// Device/Application/visualization/baseModule/grd
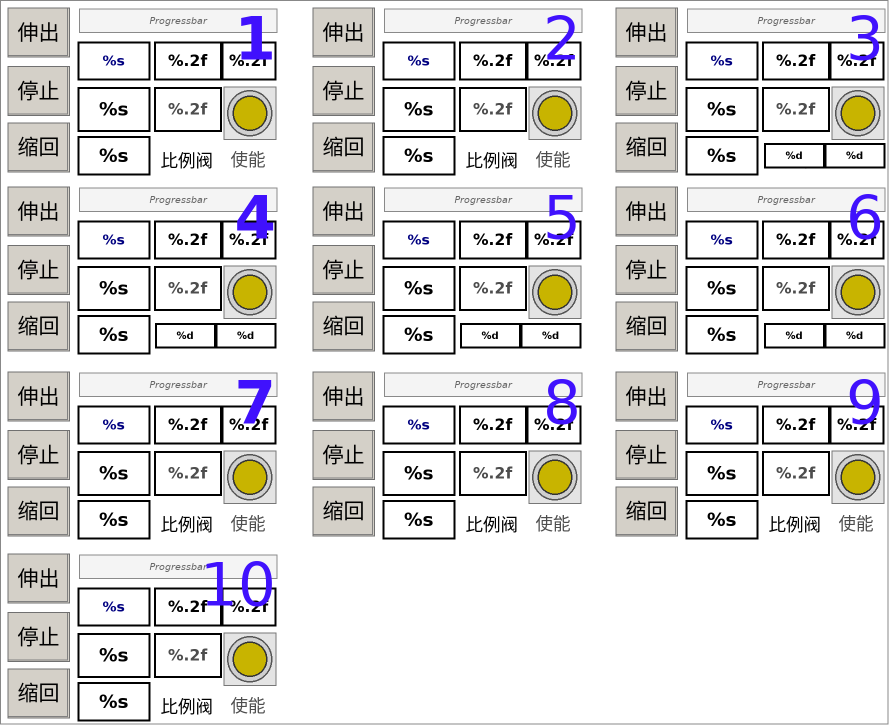
VISUALIZATION grd  // 889x725
    Frame (0,0 279x177), "1"
        shows DevUnit0(extendButton := gUI.grd[1].btnExtend, retractButton := gUI.grd[1].btnRetract, stopButton := gUI.grd[1].btnStop, percentShow := gUI.grd[1].extendPercent, nameShow := gUI.grd[1].name, wnameShow := gUI.grd[1].wname, hzname := gUI.grd[1].hzname, posShow := gUI.grd[1].postion, spdShow := gUI.grd[1].speed, pwrEnable := gUI.grd[1].pwrEnable, pwrPct := gUI.grd[1].pwrPercent)
    Frame (305,0 279x177), "2"
        shows DevUnit0(extendButton := gUI.grd[2].btnExtend, retractButton := gUI.grd[2].btnRetract, stopButton := gUI.grd[2].btnStop, percentShow := gUI.grd[2].extendPercent, nameShow := gUI.grd[2].name, wnameShow := gUI.grd[2].wname, hzname := gUI.grd[2].hzname, posShow := gUI.grd[2].postion, spdShow := gUI.grd[2].speed, pwrEnable := gUI.grd[2].pwrEnable, pwrPct := gUI.grd[2].pwrPercent)
    Frame (608,0 279x177), "3"
        shows DevUnit0(extendButton := gUI.grd[3].btnExtend, retractButton := gUI.grd[3].btnRetract, stopButton := gUI.grd[3].btnStop, percentShow := gUI.grd[3].extendPercent, nameShow := gUI.grd[3].name, wnameShow := gUI.grd[3].wname, hzname := gUI.grd[3].hzname, posShow := gUI.grd[3].postion, spdShow := gUI.grd[3].speed, pwrEnable := gUI.grd[3].pwrEnable, pwrPct := gUI.grd[3].pwrPercent)
    Frame (0,179 279x177), "4"
        shows DevUnit0(extendButton := gUI.grd[4].btnExtend, retractButton := gUI.grd[4].btnRetract, stopButton := gUI.grd[4].btnStop, percentShow := gUI.grd[4].extendPercent, nameShow := gUI.grd[4].name, wnameShow := gUI.grd[4].wname, hzname := gUI.grd[4].hzname, posShow := gUI.grd[4].postion, spdShow := gUI.grd[4].speed, pwrEnable := gUI.grd[4].pwrEnable, pwrPct := gUI.grd[4].pwrPercent)
    Frame (305,179 279x177), "5"
        shows DevUnit0(extendButton := gUI.grd[5].btnExtend, retractButton := gUI.grd[5].btnRetract, stopButton := gUI.grd[5].btnStop, percentShow := gUI.grd[5].extendPercent, nameShow := gUI.grd[5].name, wnameShow := gUI.grd[5].wname, hzname := gUI.grd[5].hzname, posShow := gUI.grd[5].postion, spdShow := gUI.grd[5].speed, pwrEnable := gUI.grd[5].pwrEnable, pwrPct := gUI.grd[5].pwrPercent)
    Frame (608,179 279x177), "6"
        shows DevUnit0(extendButton := gUI.grd[6].btnExtend, retractButton := gUI.grd[6].btnRetract, stopButton := gUI.grd[6].btnStop, percentShow := gUI.grd[6].extendPercent, nameShow := gUI.grd[6].name, wnameShow := gUI.grd[6].wname, hzname := gUI.grd[6].hzname, posShow := gUI.grd[6].postion, spdShow := gUI.grd[6].speed, pwrEnable := gUI.grd[6].pwrEnable, pwrPct := gUI.grd[6].pwrPercent)
    Frame (0,364 279x177), "7"
        shows DevUnit0(extendButton := gUI.grd[7].btnExtend, retractButton := gUI.grd[7].btnRetract, stopButton := gUI.grd[7].btnStop, percentShow := gUI.grd[7].extendPercent, nameShow := gUI.grd[7].name, wnameShow := gUI.grd[7].wname, hzname := gUI.grd[7].hzname, posShow := gUI.grd[7].postion, spdShow := gUI.grd[7].speed, pwrEnable := gUI.grd[7].pwrEnable, pwrPct := gUI.grd[7].pwrPercent)
    Frame (305,364 279x177), "8"
        shows DevUnit0(extendButton := gUI.grd[8].btnExtend, retractButton := gUI.grd[8].btnRetract, stopButton := gUI.grd[8].btnStop, percentShow := gUI.grd[8].extendPercent, nameShow := gUI.grd[8].name, wnameShow := gUI.grd[8].wname, hzname := gUI.grd[8].hzname, posShow := gUI.grd[8].postion, spdShow := gUI.grd[8].speed, pwrEnable := gUI.grd[8].pwrEnable, pwrPct := gUI.grd[8].pwrPercent)
    Frame (608,364 279x177), "9"
        shows DevUnit0(extendButton := gUI.grd[9].btnExtend, retractButton := gUI.grd[9].btnRetract, stopButton := gUI.grd[9].btnStop, percentShow := gUI.grd[9].extendPercent, nameShow := gUI.grd[9].name, wnameShow := gUI.grd[9].wname, hzname := gUI.grd[9].hzname, posShow := gUI.grd[9].postion, spdShow := gUI.grd[9].speed, pwrEnable := gUI.grd[9].pwrEnable, pwrPct := gUI.grd[9].pwrPercent)
    Frame (0,546 279x177), "10"
        shows DevUnit0(extendButton := gUI.grd[10].btnExtend, retractButton := gUI.grd[10].btnRetract, stopButton := gUI.grd[10].btnStop, percentShow := gUI.grd[10].extendPercent, nameShow := gUI.grd[10].name, wnameShow := gUI.grd[10].wname, hzname := gUI.grd[10].hzname, posShow := gUI.grd[10].postion, spdShow := gUI.grd[10].speed, pwrEnable := gUI.grd[10].pwrEnable, pwrPct := gUI.grd[10].pwrPercent)
    Frame (764,143 123x27)
        shows currentUnit(Ixt := gDev.grd[3].current[1], Irt := gDev.grd[3].current[2])
    Frame (155,323 123x27)
        shows currentUnit(Ixt := gDev.grd[4].current[1], Irt := gDev.grd[4].current[2])
    Frame (460,323 123x27)
        shows currentUnit(Ixt := gDev.grd[5].current[1], Irt := gDev.grd[5].current[2])
    Frame (764,323 123x27)
        shows currentUnit(Ixt := gDev.grd[6].current[1], Irt := gDev.grd[6].current[2])
END_VISUALIZATION

// Device/Application/visualization/baseModule/setting
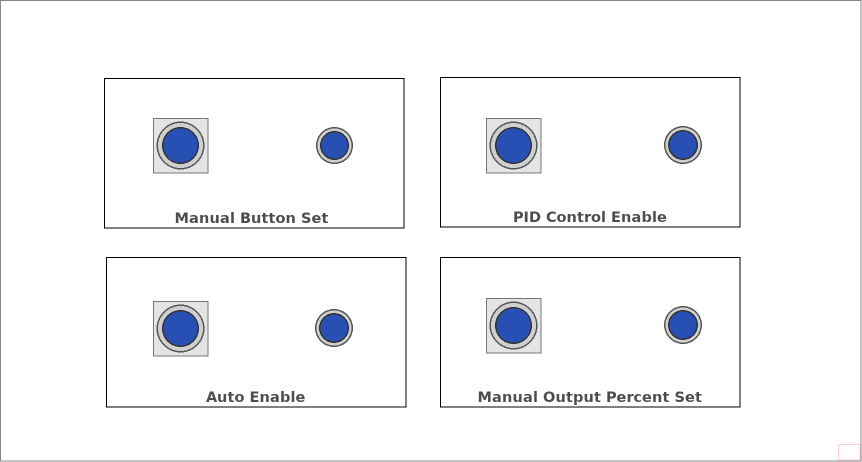
VISUALIZATION setting  // 862x462
    Rectangle (104,78 300x150), "Manual Button Set"
    Lamp1 (313,122 43x47), variable: gUI.mode.manualButtonSet, style: Lamp-Lamp1-Blue
    PushSwitchLed (153,113 55x65), variable: gUI.mode.manualButtonSet, behaviour: TOGGLE, style: Switch-PushSwitchLed-Blue
    Rectangle (440,77 300x150), "PID Control Enable"
    Lamp1 (661,122 44x46), variable: gUI.mode.usePID, style: Lamp-Lamp1-Blue
    PushSwitchLed (486,113 55x65), variable: gUI.mode.usePID, behaviour: TOGGLE, style: Switch-PushSwitchLed-Blue
    Rectangle (838,444 22x16)
    Group (106,257 300x150)
        Rectangle (0,0 300x150), "Auto Enable"
        Lamp1 (206,48 44x46), variable: gUI.mode.autoEnable, style: Lamp-Lamp1-Blue
        PushSwitchLed (47,39 55x65), variable: gUI.mode.autoEnable, behaviour: TOGGLE, style: Switch-PushSwitchLed-Blue
    Rectangle (440,257 300x150), "Manual Output Percent Set"
    Lamp1 (661,302 44x46), variable: gUI.mode.manualPercentSet, style: Lamp-Lamp1-Blue
    PushSwitchLed (486,293 55x65), variable: gUI.mode.manualPercentSet, behaviour: TOGGLE, style: Switch-PushSwitchLed-Blue
END_VISUALIZATION

// Device/Application/main
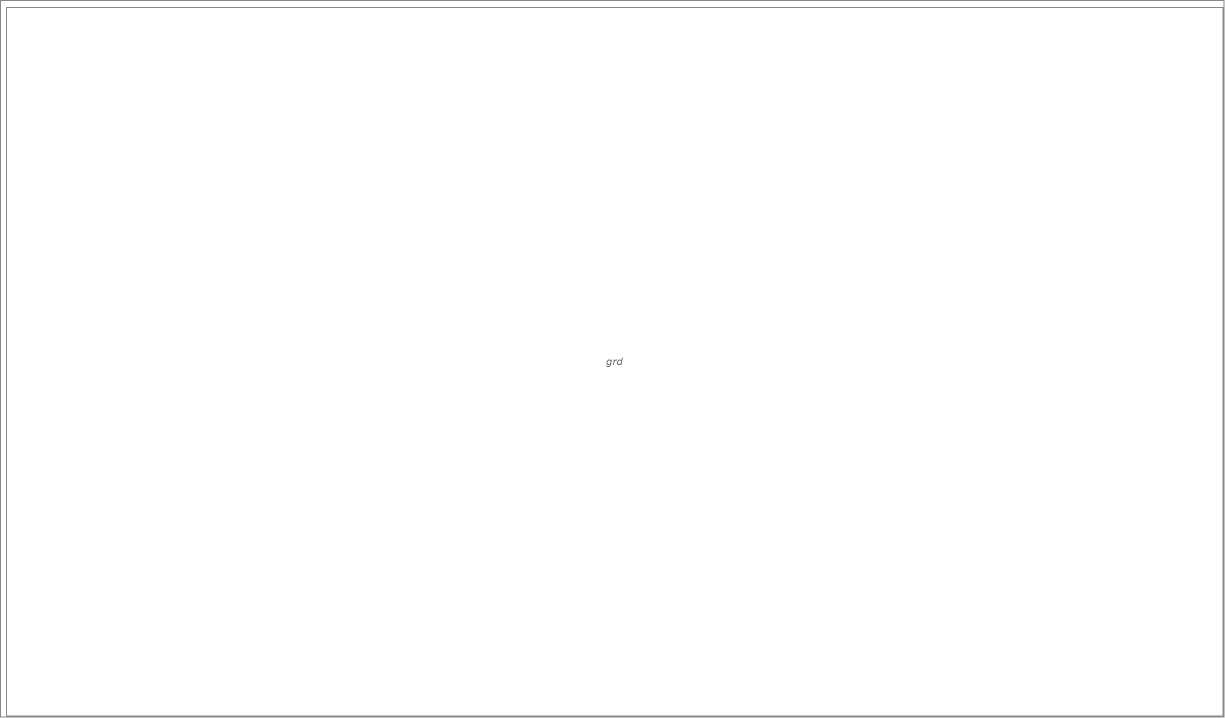
VISUALIZATION main  // 1225x718
    TabControl (6,7 1217x709)
        shows grd()
        shows sky()
        shows testPID()
        shows setting()
        [0]: ImageId=__VisualizationStyle.Element-Switch-PushSwitch-Green-On
        [1]: ImageId=__VisualizationStyle.Element-Switch-PushSwitch-Blue-On
        [2]: ImageId=__VisualizationStyle.Element-Switch-RotarySwitch-Blue-RightUp
        [3]: ImageId=__VisualizationStyle.Element-Switch-PushSwitch-Blue-On
END_VISUALIZATION

// Device/Application/visualization/baseModule/sky
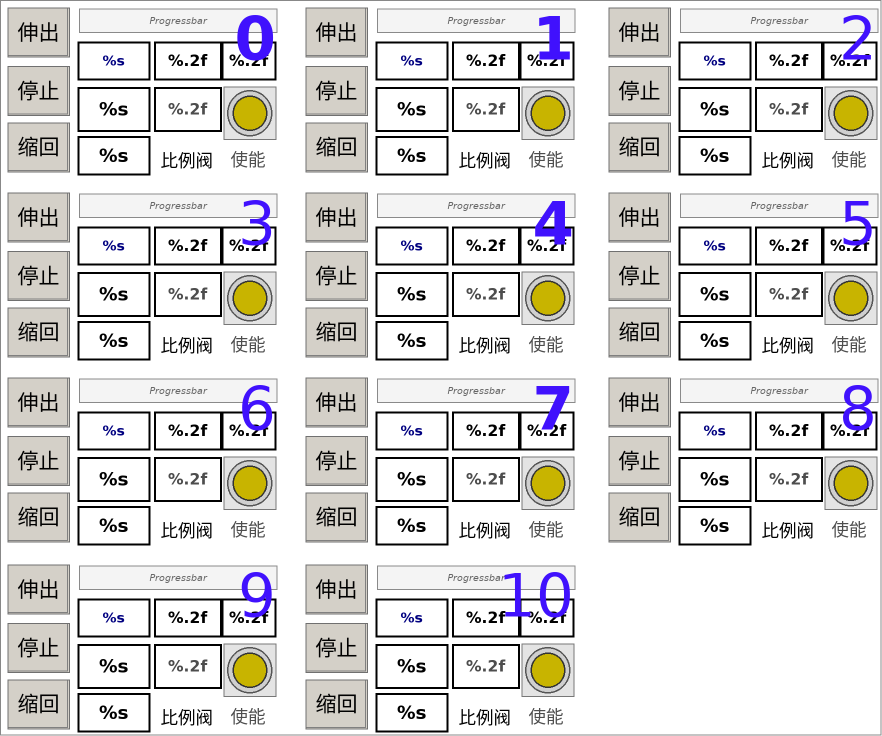
VISUALIZATION sky  // 882x736
    Frame (0,185 279x177), "3"
        shows DevUnit0(extendButton := gUI.sky[3].btnExtend, retractButton := gUI.sky[3].btnRetract, stopButton := gUI.sky[3].btnStop, percentShow := gUI.sky[3].extendPercent, nameShow := gUI.sky[3].name, wnameShow := gUI.sky[3].wname, hzname := gUI.sky[3].hzname, posShow := gUI.sky[3].postion, spdShow := gUI.sky[3].speed, pwrEnable := gUI.sky[3].pwrEnable, pwrPct := gUI.sky[3].pwrPercent)
    Frame (298,185 279x177), "4"
        shows DevUnit0(extendButton := gUI.sky[4].btnExtend, retractButton := gUI.sky[4].btnRetract, stopButton := gUI.sky[4].btnStop, percentShow := gUI.sky[4].extendPercent, nameShow := gUI.sky[4].name, wnameShow := gUI.sky[4].wname, hzname := gUI.sky[4].hzname, posShow := gUI.sky[4].postion, spdShow := gUI.sky[4].speed, pwrEnable := gUI.sky[4].pwrEnable, pwrPct := gUI.sky[4].pwrPercent)
    Frame (601,185 279x177), "5"
        shows DevUnit0(extendButton := gUI.sky[5].btnExtend, retractButton := gUI.sky[5].btnRetract, stopButton := gUI.sky[5].btnStop, percentShow := gUI.sky[5].extendPercent, nameShow := gUI.sky[5].name, wnameShow := gUI.sky[5].wname, hzname := gUI.sky[5].hzname, posShow := gUI.sky[5].postion, spdShow := gUI.sky[5].speed, pwrEnable := gUI.sky[5].pwrEnable, pwrPct := gUI.sky[5].pwrPercent)
    Frame (0,370 279x177), "6"
        shows DevUnit0(extendButton := gUI.sky[6].btnExtend, retractButton := gUI.sky[6].btnRetract, stopButton := gUI.sky[6].btnStop, percentShow := gUI.sky[6].extendPercent, nameShow := gUI.sky[6].name, wnameShow := gUI.sky[6].wname, hzname := gUI.sky[6].hzname, posShow := gUI.sky[6].postion, spdShow := gUI.sky[6].speed, pwrEnable := gUI.sky[6].pwrEnable, pwrPct := gUI.sky[6].pwrPercent)
    Frame (298,370 279x177), "7"
        shows DevUnit0(extendButton := gUI.sky[7].btnExtend, retractButton := gUI.sky[7].btnRetract, stopButton := gUI.sky[7].btnStop, percentShow := gUI.sky[7].extendPercent, nameShow := gUI.sky[7].name, wnameShow := gUI.sky[7].wname, hzname := gUI.sky[7].hzname, posShow := gUI.sky[7].postion, spdShow := gUI.sky[7].speed, pwrEnable := gUI.sky[7].pwrEnable, pwrPct := gUI.sky[7].pwrPercent)
    Frame (601,370 279x177), "8"
        shows DevUnit0(extendButton := gUI.sky[8].btnExtend, retractButton := gUI.sky[8].btnRetract, stopButton := gUI.sky[8].btnStop, percentShow := gUI.sky[8].extendPercent, nameShow := gUI.sky[8].name, wnameShow := gUI.sky[8].wname, hzname := gUI.sky[8].hzname, posShow := gUI.sky[8].postion, spdShow := gUI.sky[8].speed, pwrEnable := gUI.sky[8].pwrEnable, pwrPct := gUI.sky[8].pwrPercent)
    Frame (0,557 279x177), "9"
        shows DevUnit0(extendButton := gUI.sky[9].btnExtend, retractButton := gUI.sky[9].btnRetract, stopButton := gUI.sky[9].btnStop, percentShow := gUI.sky[9].extendPercent, nameShow := gUI.sky[9].name, wnameShow := gUI.sky[9].wname, hzname := gUI.sky[9].hzname, posShow := gUI.sky[9].postion, spdShow := gUI.sky[9].speed, pwrEnable := gUI.sky[9].pwrEnable, pwrPct := gUI.sky[9].pwrPercent)
    Frame (298,557 279x177), "10"
        shows DevUnit0(extendButton := gUI.sky[10].btnExtend, retractButton := gUI.sky[10].btnRetract, stopButton := gUI.sky[10].btnStop, percentShow := gUI.sky[10].extendPercent, nameShow := gUI.sky[10].name, wnameShow := gUI.sky[10].wname, hzname := gUI.sky[10].hzname, posShow := gUI.sky[10].postion, spdShow := gUI.sky[10].speed, pwrEnable := gUI.sky[10].pwrEnable, pwrPct := gUI.sky[10].pwrPercent)
    Frame (298,0 279x177), "1"
        shows DevUnit0(extendButton := gUI.sky[1].btnExtend, retractButton := gUI.sky[1].btnRetract, stopButton := gUI.sky[1].btnStop, percentShow := gUI.sky[1].extendPercent, nameShow := gUI.sky[1].name, wnameShow := gUI.sky[1].wname, hzname := gUI.sky[1].hzname, posShow := gUI.sky[1].postion, spdShow := gUI.sky[1].speed, pwrEnable := gUI.sky[1].pwrEnable, pwrPct := gUI.sky[1].pwrPercent)
    Frame (601,0 279x177), "2"
        shows DevUnit0(extendButton := gUI.sky[2].btnExtend, retractButton := gUI.sky[2].btnRetract, stopButton := gUI.sky[2].btnStop, percentShow := gUI.sky[2].extendPercent, nameShow := gUI.sky[2].name, wnameShow := gUI.sky[2].wname, hzname := gUI.sky[2].hzname, posShow := gUI.sky[2].postion, spdShow := gUI.sky[2].speed, pwrEnable := gUI.sky[2].pwrEnable, pwrPct := gUI.sky[2].pwrPercent)
    Frame (0,0 279x177), "0"
        shows DevUnit0(extendButton := gUI.sky[0].btnExtend, retractButton := gUI.sky[0].btnRetract, stopButton := gUI.sky[0].btnStop, percentShow := gUI.sky[0].extendPercent, nameShow := gUI.sky[0].name, wnameShow := gUI.sky[0].wname, hzname := gUI.sky[0].hzname, posShow := gUI.sky[0].postion, spdShow := gUI.sky[0].speed, pwrEnable := gUI.sky[0].pwrEnable, pwrPct := gUI.sky[0].pwrPercent)
END_VISUALIZATION

// Device/Application/visualization/baseModule/BasePID
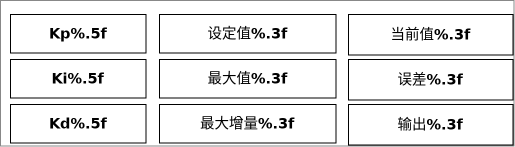
VISUALIZATION BasePID  // 515x147
VAR_IN_OUT
	pid_Kp			:REAL;
	pid_Ki  		:REAL;
	pid_Kd			:REAL;
	pid_Set_Val		:REAL;
	pid_Max_Val		:REAL;
	pid_Max_Acc		:REAL;
	Pid_Act_Val		:REAL;
	Pid_Out			:REAL;
	Pid_Err			:REAL;

END_VAR
    RoundedRectangle (10,14 136x39), "Kp%.5f", text variable: pid_Kp
        OnMouseDown: write the text variable via Default, min 0
    RoundedRectangle (10,59 136x39), "Ki%.5f", text variable: pid_Ki
        OnMouseDown: write the text variable via Default, min 0
    RoundedRectangle (10,104 136x39), "Kd%.5f", text variable: pid_Kd
        OnMouseDown: write the text variable via Default, min 0
    RoundedRectangle (159,14 177x39), "设定值%.3f", text variable: pid_Set_Val
        OnMouseDown: write the text variable via Default
    RoundedRectangle (159,59 177x39), "最大值%.3f", text variable: pid_Max_Val
        OnMouseDown: write the text variable via Default
    RoundedRectangle (159,104 177x39), "最大增量%.3f", text variable: pid_Max_ACC
        OnMouseDown: write the text variable via Default
    RoundedRectangle (348,14 165x41), "当前值%.3f", text variable: Pid_Act_Val
    RoundedRectangle (348,59 165x41), "误差%.3f", text variable: Pid_Err
    RoundedRectangle (348,104 165x41), "输出%.3f", text variable: Pid_Out
END_VISUALIZATION

// Device/Application/visualization/baseModule/testPID
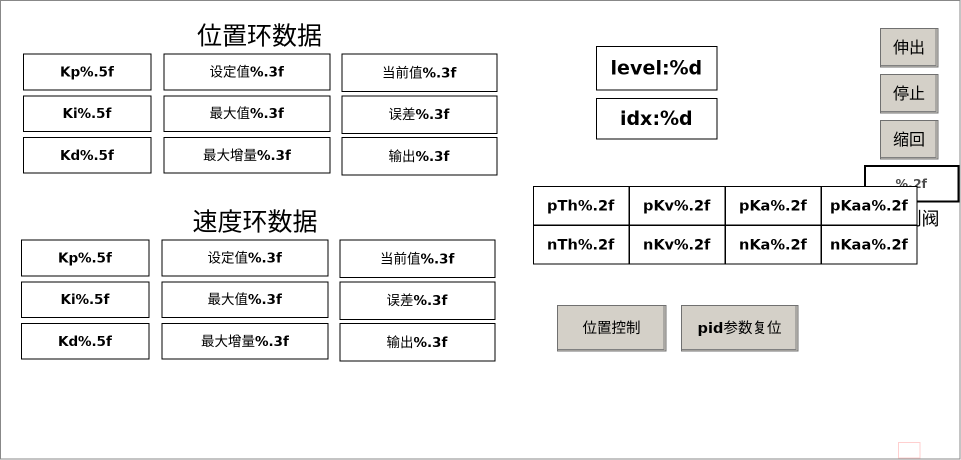
VISUALIZATION testPID  // 961x460
    Frame (14,41 485x136)
        shows BasePID(pid_Kp := gUI.pid.pos.Kp, pid_Ki := gUI.pid.pos.Ki, pid_Kd := gUI.pid.pos.Kd, pid_Set_Val := gUI.pid.pos.Set_Point, pid_Max_Val := gUI.pid.pos.Max_Val, pid_Max_Acc := gUI.pid.pos.Max_ACC, Pid_Act_Val := gUI.pid.pos.Act_Val, Pid_Out := gUI.pid.pos.OUT, Pid_Err := gUI.pid.pos.Err)
    Label (101,15 317x41), "位置环数据"
    Label (107,201 296x41), "速度环数据"
    Frame (12,227 485x136)
        shows BasePID(pid_Kp := gUI.pid.spd.Kp, pid_Ki := gUI.pid.spd.Ki, pid_Kd := gUI.pid.spd.Kd, pid_Set_Val := gUI.pid.spd.Set_Point, pid_Max_Val := gUI.pid.spd.Max_Val, pid_Max_Acc := gUI.pid.spd.Max_ACC, Pid_Act_Val := gUI.pid.spd.Act_Val, Pid_Out := gUI.pid.spd.OUT, Pid_Err := gUI.pid.spd.Err)
    Group (596,46 121x93)
        RoundedRectangle (0,52 121x41), "idx:%d", text variable: gUI.pid.idx
            OnMouseDown: write the text variable via Default, min 0, max 10
        RoundedRectangle (0,0 121x44), "level:%d", text variable: gUI.pid.level
            OnMouseDown: write the text variable via Default, min 1, max 2
    Button (557,305 109x46), "位置控制"
        toggle gUI.pid.posBtn
    Rectangle (898,442 22x16)
    Group (864,28 55x133)
        Button (16,92 58x39), "缩回"
            toggle gUI.pid.retractBtn
        Button (16,46 58x39), "停止"
            toggle gUI.pid.stopBtn
        Button (16,0 58x39), "伸出"
            toggle gUI.pid.extendBtn
        Group (0,137 95x68)
            RoundedRectangle (0,0 95x37), "%.2f", text variable: gUI.pid.pwrPercent
                OnMouseDown: write the text variable via Default, min 0, max 100
            Label (10,40 77x28), "比例阀"
    Button (681,305 117x46), "pid参数复位"
        tap gUI.pid.rstPidBtn
    Group (533,186 384x78)
        RoundedRectangle (0,0 96x39), "pTh%.2f", text variable: gUI.pid.ff.pstThreshold
            OnMouseDown: write the text variable via Default, min 0
        RoundedRectangle (0,39 96x39), "nTh%.2f", text variable: gUI.pid.ff.negThreshold
            OnMouseDown: write the text variable via Default, min 0
        RoundedRectangle (96,0 96x39), "pKv%.2f", text variable: gUI.pid.ff.pstKv
            OnMouseDown: write the text variable via Default, min 0
        RoundedRectangle (192,0 96x39), "pKa%.2f", text variable: gUI.pid.ff.pstKa
            OnMouseDown: write the text variable via Default, min 0
        RoundedRectangle (288,0 96x39), "pKaa%.2f", text variable: gUI.pid.ff.pstKaa
            OnMouseDown: write the text variable via Default, min 0
        RoundedRectangle (96,39 96x39), "nKv%.2f", text variable: gUI.pid.ff.negKv
            OnMouseDown: write the text variable via Default, min 0
        RoundedRectangle (192,39 96x39), "nKa%.2f", text variable: gUI.pid.ff.negKa
            OnMouseDown: write the text variable via Default, min 0
        RoundedRectangle (288,39 96x39), "nKaa%.2f", text variable: gUI.pid.ff.negKaa
            OnMouseDown: write the text variable via Default, min 0
END_VISUALIZATION

// Device/Application/visualization/baseModule/currentUnit
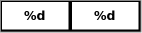
VISUALIZATION currentUnit  // 142x33
VAR_IN_OUT
	Ixt		:	WORD;
	Irt		:	WORD;
END_VAR
    RoundedRectangle (0,0 70x31), "%d", text variable: Ixt
    RoundedRectangle (70,0 70x31), "%d", text variable: Irt
END_VISUALIZATION
